// TIA Portal V21 export
// export: Created 2026-06-08T03:11:54.7246491Z, ExportSetting WithReadOnly, DisplayName Totally Integrated Automation Portal, DisplayVersion V21, DisplayName SINAMICS Startdrive Advanced, DisplayVersion V21, DisplayName SINAMICS Startdrive G110M, G120, G120C, G120D, G120P, G115D, DisplayVersion V21, DisplayName SINAMICS Startdrive G130, G150, S120, S150, G200, G220, S200, S210, S220, Innomotics MVD, DisplayVersion V21, DisplayName STEP 7 Professional, DisplayVersion V21, DisplayName STEP 7 Safety, DisplayVersion V21, DisplayName Tech WebApplication, DisplayVersion V21, DisplayName WinCC Basic/Comfort/Advanced, DisplayVersion V21, DisplayName WinCC Professional, DisplayVersion V21, DisplayName WinCC Unified, DisplayVersion V21
FUNCTION_BLOCK "FB_CommsWatchdog_LAD"   // FB3, LAD
TITLE = Heartbeat changed
{ S7_Optimized_Access := 'TRUE' }
// stored: CodeModifiedDate 2026-06-08T03:10:14.5196473Z, CompileDate 2026-06-08T03:11:41.0634515Z, CreationDate 2026-06-08T03:07:13.4993738Z, DownloadDate 0001-01-01T00:00:00Z, InterfaceModifiedDate 2026-06-08T03:10:14.5196473Z, IsConsistent true, LibraryConformanceStatus 该对象为库兼容。, LoadMemoryLength 4239, MemoryReserve 100, ModifiedDate 2026-06-08T03:10:27.490681Z, PLCSimAdvancedSupport true, ParameterModified 2026-06-08T03:09:18.1248756Z, SetENOAutomatically false, StructureModified 2026-06-08T03:10:14.5196473Z, WorkMemoryLength 18
   VAR_INPUT
      Remote_Heartbeat : Int;
   END_VAR
   VAR_OUTPUT
      Remote_Comms_OK : Bool;
      Watchdog_Timer : Int;
   END_VAR
   VAR
      Last_Heartbeat : Int;
      Heartbeat_Changed : Bool;
      tWatchdog : TON_TIME;
   END_VAR
BEGIN
END_FUNCTION_BLOCK
